(*
SPDX-FileCopyrightText: © 2026 Oleksandr Tiutyk <trofimich@gmail.com>
SPDX-License-Identifier: MIT
License: https://opensource.org/license/mit
*)

(*!
<summary>
Beckhoff EL2008: 8-channel digital output terminal (24 V DC, 0.5 A).
</summary>
<description>
Process image mapping structure for the EL2008 EtherCAT terminal with 8 discrete 24 V DC 0.5 A outputs.
When used for I/O, link located fields or their containing buffers to the matching selected PDOs.
The record is not a packed wire buffer; compiler padding is not part of the device specification.
Unlinked/default values do not prove valid I/O. The caller evaluates bus/channel validity before use.
Use one owner task per instance and externally synchronize other access; multi-field snapshots are not atomic.
Copies store data without creating hardware links. Keep borrowed field references valid while consumers are bound.
This passive record performs no validation, synchronization, configuration or protocol advancement.
</description>
*)
TYPE EL2008 :
STRUCT
	Ch1 AT %Q* : BOOL;
	Ch2 AT %Q* : BOOL;
	Ch3 AT %Q* : BOOL;
	Ch4 AT %Q* : BOOL;
	Ch5 AT %Q* : BOOL;
	Ch6 AT %Q* : BOOL;
	Ch7 AT %Q* : BOOL;
	Ch8 AT %Q* : BOOL;
END_STRUCT
END_TYPE

(* stored: Version 1.1.0.1, ProductVersion 3.1.4026.20
   DUT EL2008: Id {a8fb9a9a-5645-4e21-bef6-2f5b45345b29} *)
